FUNCTION_BLOCK SWITCH (* Switch(demultiplex)an event *)
  (* Standard: 61499-1 *)
  (* Version 7.0, 01/12/2011, LAPAS, UDESC *)
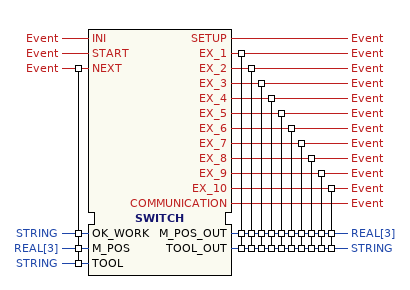
  EVENT_INPUT
    INI; (* Inicializa o bloco *)
    START; (* Inicia o primeiro evento de saida *)
    NEXT WITH OK_WORK, M_POS, TOOL; (* Gera o proximo evento de saida *)
  END_EVENT
  EVENT_OUTPUT
    SETUP; (* Setup da maquina *)
    EX_1 WITH M_POS_OUT, TOOL_OUT; (* Executable 1 *)
    EX_2 WITH M_POS_OUT, TOOL_OUT; (* Executable 2 *)
    EX_3 WITH M_POS_OUT, TOOL_OUT; (* Executable 3 *)
    EX_4 WITH M_POS_OUT, TOOL_OUT; (* Executable 4 *)
    EX_5 WITH M_POS_OUT, TOOL_OUT; (* Executable 5 *)
    EX_6 WITH M_POS_OUT, TOOL_OUT; (* Executable 6 *)
    EX_7 WITH M_POS_OUT, TOOL_OUT; (* Executable 7 *)
    EX_8 WITH M_POS_OUT, TOOL_OUT; (* Executable 8 *)
    EX_9 WITH M_POS_OUT, TOOL_OUT; (* Executable 9 *)
    EX_10 WITH M_POS_OUT, TOOL_OUT; (* Executable 10 *)
    COMMUNICATION; (* comunicacao *)
  END_EVENT
  VAR_INPUT
    OK_WORK : STRING;
    M_POS : ARRAY [0..2] OF REAL;
    TOOL : STRING;
  END_VAR
  VAR_OUTPUT
    M_POS_OUT : ARRAY [0..2] OF REAL;
    TOOL_OUT : STRING;
  END_VAR
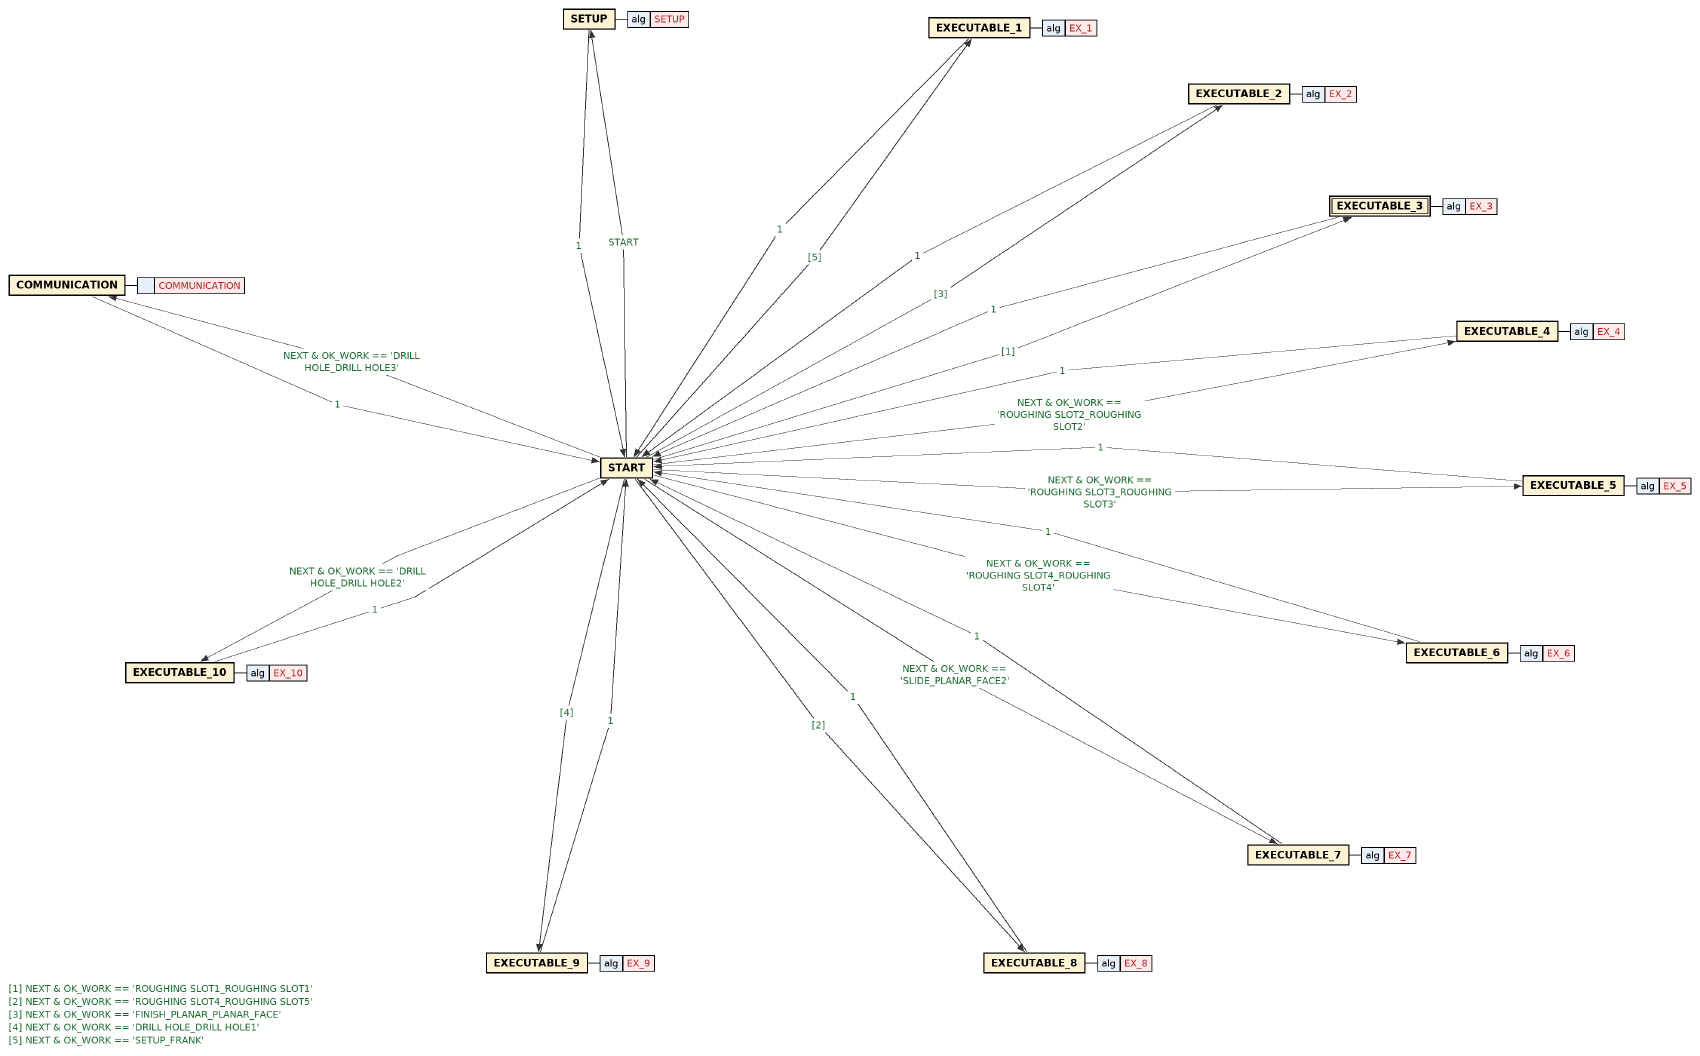
  EC_STATES
    EXECUTABLE_3 : alg -> EX_3;
    EXECUTABLE_6 : alg -> EX_6;
    EXECUTABLE_5 : alg -> EX_5;
    EXECUTABLE_4 : alg -> EX_4;
    EXECUTABLE_8 : alg -> EX_8;
    START;
    EXECUTABLE_7 : alg -> EX_7;
    COMMUNICATION : -> COMMUNICATION;
    EXECUTABLE_2 : alg -> EX_2;
    EXECUTABLE_1 : alg -> EX_1;
    EXECUTABLE_9 : alg -> EX_9;
    SETUP : alg -> SETUP;
    EXECUTABLE_10 : alg -> EX_10;
  END_STATES
  EC_TRANSITIONS
    START TO SETUP := START;
    START TO EXECUTABLE_1 := NEXT & OK_WORK == 'SETUP_FRANK';
    START TO EXECUTABLE_2 := NEXT & OK_WORK == 'FINISH_PLANAR_PLANAR_FACE';
    START TO EXECUTABLE_3 := NEXT & OK_WORK == 'ROUGHING SLOT1_ROUGHING SLOT1';
    START TO EXECUTABLE_4 := NEXT & OK_WORK == 'ROUGHING SLOT2_ROUGHING SLOT2';
    START TO EXECUTABLE_5 := NEXT & OK_WORK == 'ROUGHING SLOT3_ROUGHING SLOT3';
    START TO EXECUTABLE_6 := NEXT & OK_WORK == 'ROUGHING SLOT4_ROUGHING SLOT4';
    START TO EXECUTABLE_7 := NEXT & OK_WORK == 'SLIDE_PLANAR_FACE2';
    START TO EXECUTABLE_8 := NEXT & OK_WORK == 'ROUGHING SLOT4_ROUGHING SLOT5';
    START TO EXECUTABLE_9 := NEXT & OK_WORK == 'DRILL HOLE_DRILL HOLE1';
    START TO EXECUTABLE_10 := NEXT & OK_WORK == 'DRILL HOLE_DRILL HOLE2';
    START TO COMMUNICATION := NEXT & OK_WORK == 'DRILL HOLE_DRILL HOLE3';
    SETUP TO START := 1;
    EXECUTABLE_1 TO START := 1;
    EXECUTABLE_2 TO START := 1;
    EXECUTABLE_3 TO START := 1;
    EXECUTABLE_4 TO START := 1;
    EXECUTABLE_5 TO START := 1;
    EXECUTABLE_6 TO START := 1;
    EXECUTABLE_7 TO START := 1;
    EXECUTABLE_8 TO START := 1;
    EXECUTABLE_9 TO START := 1;
    EXECUTABLE_10 TO START := 1;
    COMMUNICATION TO START := 1;
  END_TRANSITIONS
  ALGORITHM alg IN Lua:
M_POS_OUT[1] = M_POS[1] M_POS_OUT[2] = M_POS[2] M_POS_OUT[3] = M_POS[3]
  END_ALGORITHM
END_FUNCTION_BLOCK
